(* PLC project stop, Dassault Systèmes ControlBuild 2024x *)
(* stored: creationDateTime 2023-10-03T11:12:55-01:00 *)

(* This module simulates the behaviour of a mechanical stop. *)
FUNCTION_BLOCK equipment_library.stop
  VAR_INPUT
    incPositionX : REAL := 0.0;
    incPositionY : REAL := 0.0;
    incPositionZ : REAL := 0.0;
  END_VAR
  VAR_INPUT
    coordCenterX : REAL := 0.0;
    coordCenterY : REAL := 0.0;
    coordCenterZ : REAL := 0.0;
    incRotationX : REAL := 0.0;
    incRotationY : REAL := 0.0;
    incRotationZ : REAL := 0.0;
  END_VAR
  VAR
    status_act_prod : DINT := 0;
    m11 : REAL := 1.0;
    m12 : REAL := 0.0;
    m13 : REAL := 0.0;
    m14 : REAL := 0.0;
    m21 : REAL := 0.0;
    m22 : REAL := 1.0;
    m23 : REAL := 0.0;
    m24 : REAL := 0.0;
    m31 : REAL := 0.0;
    m32 : REAL := 0.0;
    m33 : REAL := 1.0;
    m34 : REAL := 0.0;
    m41 : REAL := 0.0;
    m42 : REAL := 0.0;
    m43 : REAL := 0.0;
    m44 : REAL := 1.0;
  END_VAR


ACTION C_source_code:
/* ----------------------------------------------------------------	*/
/* Type : Model of Operative Behaviour					*/
/* Category :  Actors and Products						*/
/* Author : Dassault Systemes						*/
/* Update date : June 2018							*/
/* ----------------------------------------------------------------	*/
/* This module simulates the behaviour of a mechanical stop.		*/
/* ----------------------------------------------------------------	*/

/* ----------------------------------------------------------------	*/
/* Shift of the stop for a 3-axes locking					*/
/* ----------------------------------------------------------------	*/
if ((incPositionX != 0.0) || (incPositionY != 0.0) || (incPositionZ != 0.0))
	moveBy(myself, incPositionX, incPositionY, incPositionZ);



/* ----------------------------------------------------------------	*/
/* Rotation of the stop when embedded on a rotary plate ring		*/
/* ----------------------------------------------------------------	*/
if ((incRotationX != 0.0) || (incRotationY != 0.0) || (incRotationZ != 0.0))
	rotateBy(myself, incRotationX, incRotationY, incRotationZ, coordCenterX, coordCenterY, coordCenterZ);
END_ACTION
END_FUNCTION_BLOCK
